TYPE MoverSort :
STRUCT
	MoverNumber : UDINT;
	TrackID : PlanarTrackOTCID;
	MoverPos : LREAL;
END_STRUCT
END_TYPE

(* stored: Version 1.1.0.1, ProductVersion 3.1.4026.8
   DUT MoverSort: Id {bdc1f80e-235a-417d-8a26-298e40606bc2} *)
